(* CoDeSys 2.3 export: ST_SE_CYLINDER_POS_CFG.EXP *)

(* Data type *)
TYPE ST_SE_CYLINDER_POS_CFG :
STRUCT
	Ease : REAL;

	TgtLS_In  : REAL;
	TgtLS_Out : REAL;
	TgtLS_Slow  : REAL;

	LS_Limit_In  : BOOL;
	LS_Limit_Out : BOOL;

	Cycle   : REAL; (*Seconds*)
	TimeEase: REAL; (*Seconds*)
	TimeMax : REAL; (*Seconds*)

	HP : BYTE;

END_STRUCT
END_TYPE
